ABB RobotStudio station: trabalho.rsstnx

Station Project6 (saved by RobotStudio 24.3.10958.1)
Controller IRB120_3_58
  mechanical unit ROB_1: IRB120_3_58__01, 6 joints, base frame (0, 0, 0) mm
Layout (positions relative to the parent item):
  - IRB120_3_58__01 [mechanism, from %ABB.RobotStudio.Models.IRB120%\IRB120_3_58_G_01.rslib] at (0, 0, 0) mm; joint values [0, 0, 0, 0, 0.5236, 0] (rad or m)
  - MyTool [mechanism, from Training Objects\myTool.rslib] at (364.35, 0, 594) mm, rotated rx 180 ry 60 rz 180 deg
  - mesa [part] at (200, -200, 0) mm, size 300 x 400 x 300 mm
  - tampa [part] at (350, 0, 380) mm, size 16 x 15 x 20 mm
  - Attacher [smart component, from Components\Attacher.rslib]
      properties: Parent=MyTool; Flange=0; Child=tampa; Mount=false; Offset=[0 0 0]; Orientation=[0 0 0]
  - Detacher [smart component, from Components\Detacher.rslib]
      properties: Child=tampa; KeepPosition=true
  - Rotator2 [smart component, from Components\Rotator2.rslib]
      properties: Object=tampa; CenterPoint=[0.35 0 0.38]; Axis=[0 0 1]; Angle=-1.5707963267949; Duration=2; Reference=Global; ReferenceObject=tampa
  - corpo [part], size 50 x 49.9 x 70 mm
  - Positioner [smart component, from Components\Positioner.rslib]
      properties: Object=tampa; Position=[0.35 0 0.38]; Orientation=[0 0 0]; Reference=Global; ReferenceObject=corpo
  - Positioner_2 [smart component, from Components\Positioner.rslib]
      properties: Object=tampa; Position=[0.35 0.11 0.32]; Orientation=[0 0 0]; Reference=Global; ReferenceObject=(none)
Attachment: MyTool is attached to IRB120_3_58__01 / Link6
Attachment: tampa is attached to MyTool / SpintecTool
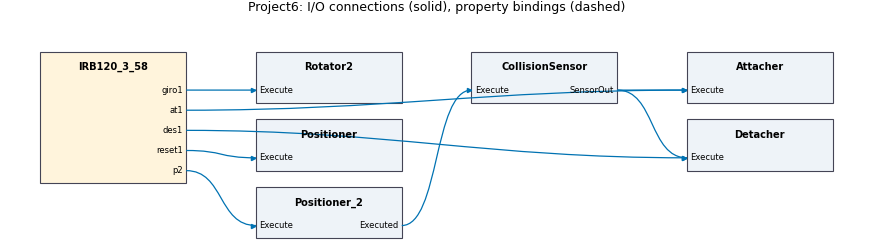
Station logic (signal -> signal, property => property):
  CollisionSensor.SensorOut -> Attacher.Execute
  CollisionSensor_2.SensorOut -> Detacher.Execute
  Positioner_2.Executed -> Rotator2_2.Execute
  IRB120_3_58.giro1 -> Rotator2.Execute
  IRB120_3_58.at1 -> Attacher.Execute
  IRB120_3_58.des1 -> Detacher.Execute
  IRB120_3_58.reset1 -> Positioner.Execute
  IRB120_3_58.p2 -> Positioner_2.Execute
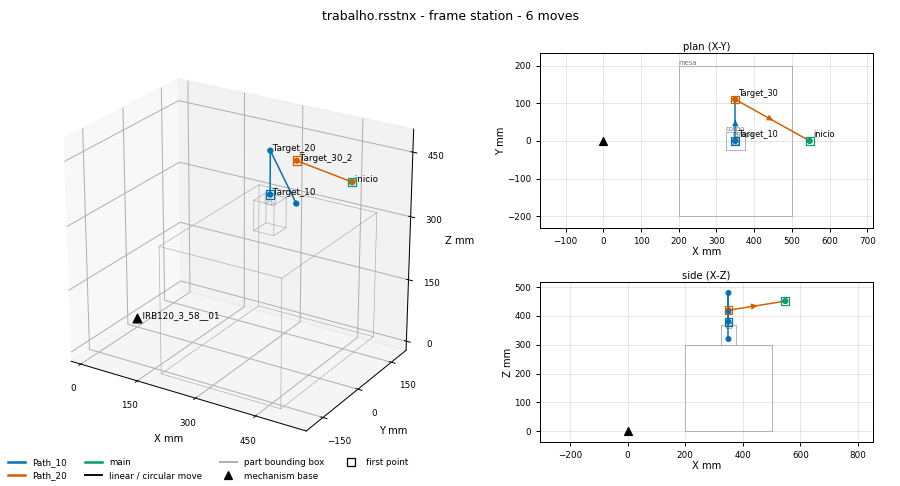
[picture p0: tool path of trabalho.rsstnx in frame station, 6 of 6 moves have a stored position in this frame; points joined in program order, loops and branches not executed]
Targets, tools, work objects and paths stored in the station, written as RAPID:
! task T_ROB1
MODULE CalibData
  PERS tooldata MyTool:=[TRUE,[[31.792631019,0,229.638935148],[0.945518576,0,0.325568154,0]],[1,[0,0,1],[1,0,0,0],0,0,0]];
ENDMODULE

! task T_ROB1
MODULE Module1
  CONST robtarget Target_10:=[[350,0,380],[0,0,1,0],[0,0,0,0],[9E+09,9E+09,9E+09,9E+09,9E+09,9E+09]];
  CONST robtarget inicio:=[[547.33065187,0,451.647288113],[0.19080896,0,0.98162719,0],[0,0,0,0],[9E+09,9E+09,9E+09,9E+09,9E+09,9E+09]];
  CONST robtarget Target_20:=[[350.000046167,0,479.999936598],[-0.000000052,0,1,0],[0,0,0,0],[9E+09,9E+09,9E+09,9E+09,9E+09,9E+09]];
  CONST robtarget Target_30:=[[350,110,320],[0,0,1,0],[0,0,0,0],[9E+09,9E+09,9E+09,9E+09,9E+09,9E+09]];
  CONST robtarget Target_30_2:=[[350,110,420],[0,0,1,0],[0,0,0,0],[9E+09,9E+09,9E+09,9E+09,9E+09,9E+09]];
  PROC Path_10()
    MoveL Target_10,v200,fine,MyTool\WObj:=wobj0;
    WaitTime 1;
    Set giro1;
    WaitTime 2.5;
    Set at1;
    MoveL Target_20,v200,fine,MyTool\WObj:=wobj0;
    MoveL Target_30,v200,fine,MyTool\WObj:=wobj0;
  ENDPROC
  PROC Path_20()
    Set des1;
    WaitTime 1;
    Set p2;
    MoveL Target_30_2,v500,z100,MyTool\WObj:=wobj0;
    MoveL inicio,v500,z100,MyTool\WObj:=wobj0;
  ENDPROC
  PROC main()
    MoveL inicio,v1000,z100,MyTool\WObj:=wobj0;
    Reset at1;
    Reset giro1;
    Reset des1;
    Reset p2;
    Reset reset1;
    WaitTime 1;
    Set reset1;
    Path_10;
    WaitTime 2;
    Path_20;
  ENDPROC
ENDMODULE

